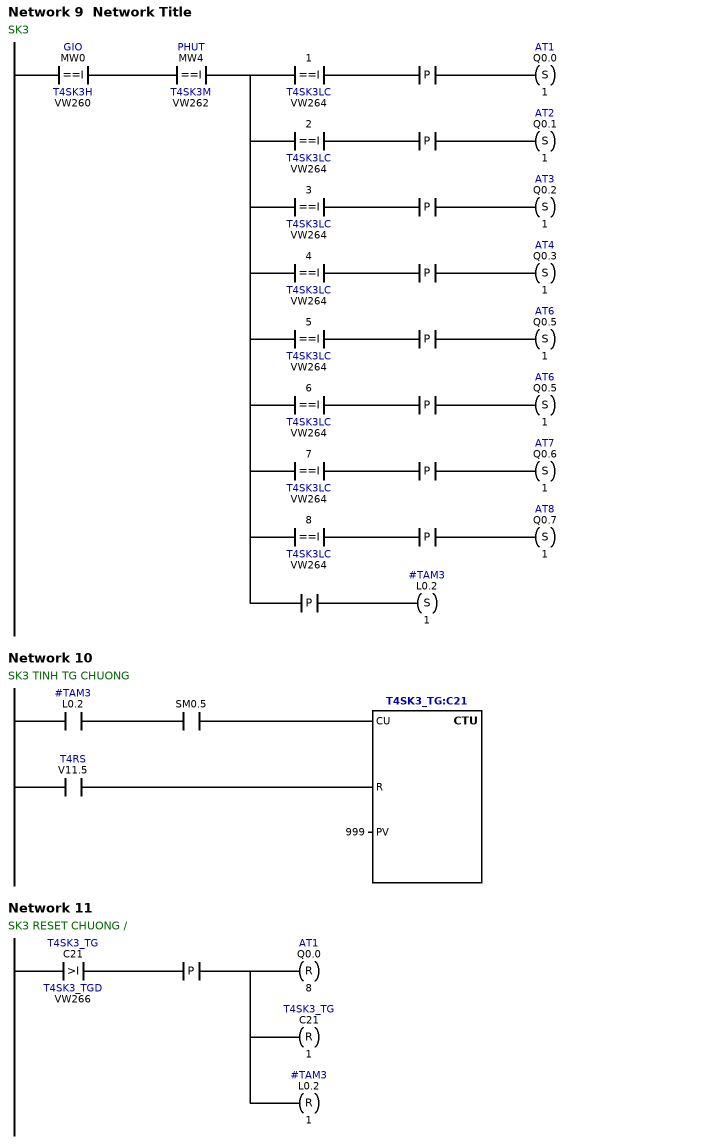
[picture p24: SBR5 networks 9-11]
Network 9 // Network Title
// SK3	
LDW=   GIO:MW0, T4SK3H:VW260
AW=    PHUT:MW4, T4SK3M:VW262
LPS
AW=    1, T4SK3LC:VW264
EU
S      AT1:Q0.0, 1
LRD
AW=    2, T4SK3LC:VW264
EU
S      AT2:Q0.1, 1
LRD
AW=    3, T4SK3LC:VW264
EU
S      AT3:Q0.2, 1
LRD
AW=    4, T4SK3LC:VW264
EU
S      AT4:Q0.3, 1
LRD
AW=    5, T4SK3LC:VW264
EU
S      AT6:Q0.5, 1
LRD
AW=    6, T4SK3LC:VW264
EU
S      AT6:Q0.5, 1
LRD
AW=    7, T4SK3LC:VW264
EU
S      AT7:Q0.6, 1
LRD
AW=    8, T4SK3LC:VW264
EU
S      AT8:Q0.7, 1
LPP
EU
S      #TAM3:L0.2, 1
Network 10
// SK3 TINH TG CHUONG
LD     #TAM3:L0.2
A      SM0.5
LD     T4RS:V11.5
CTU    T4SK3_TG:C21, 999
Network 11
// SK3 RESET CHUONG
// 
LDW>   T4SK3_TG:C21, T4SK3_TGD:VW266
EU
R      AT1:Q0.0, 8
R      T4SK3_TG:C21, 1
R      #TAM3:L0.2, 1
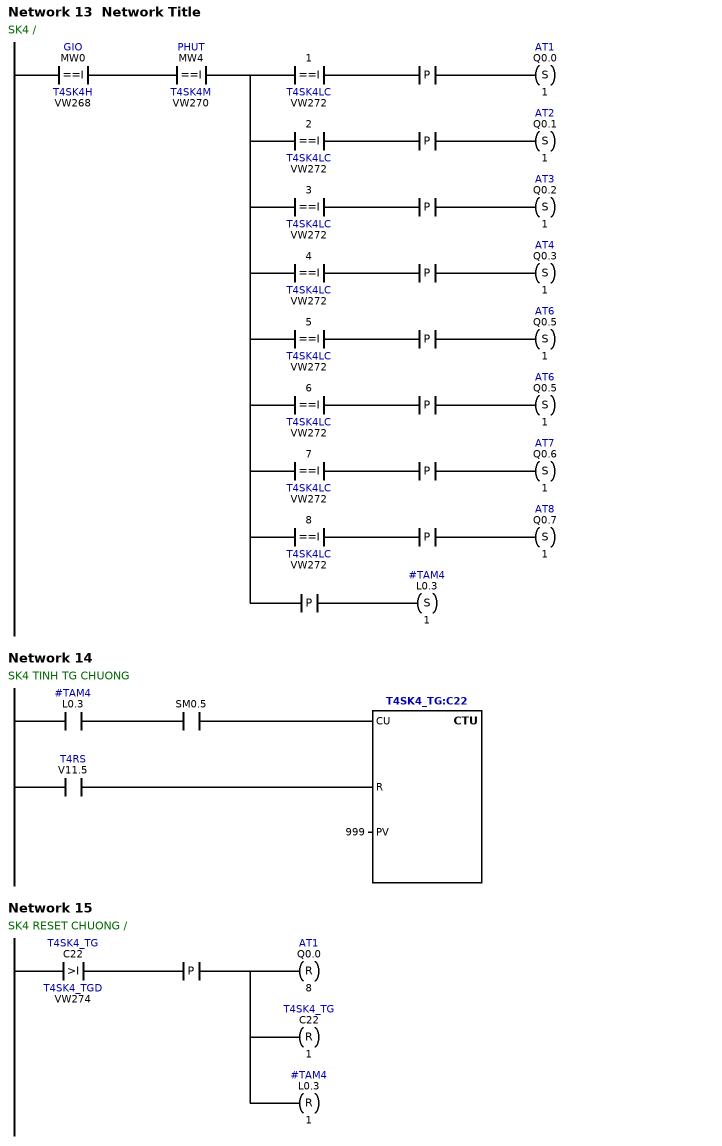
Network 13 // Network Title
// SK4
// 	
LDW=   GIO:MW0, T4SK4H:VW268
AW=    PHUT:MW4, T4SK4M:VW270
LPS
AW=    1, T4SK4LC:VW272
EU
S      AT1:Q0.0, 1
LRD
AW=    2, T4SK4LC:VW272
EU
S      AT2:Q0.1, 1
LRD
AW=    3, T4SK4LC:VW272
EU
S      AT3:Q0.2, 1
LRD
AW=    4, T4SK4LC:VW272
EU
S      AT4:Q0.3, 1
LRD
AW=    5, T4SK4LC:VW272
EU
S      AT6:Q0.5, 1
LRD
AW=    6, T4SK4LC:VW272
EU
S      AT6:Q0.5, 1
LRD
AW=    7, T4SK4LC:VW272
EU
S      AT7:Q0.6, 1
LRD
AW=    8, T4SK4LC:VW272
EU
S      AT8:Q0.7, 1
LPP
EU
S      #TAM4:L0.3, 1
Network 14
// SK4 TINH TG CHUONG
LD     #TAM4:L0.3
A      SM0.5
LD     T4RS:V11.5
CTU    T4SK4_TG:C22, 999
Network 15
// SK4 RESET CHUONG
// 
LDW>   T4SK4_TG:C22, T4SK4_TGD:VW274
EU
R      AT1:Q0.0, 8
R      T4SK4_TG:C22, 1
R      #TAM4:L0.3, 1
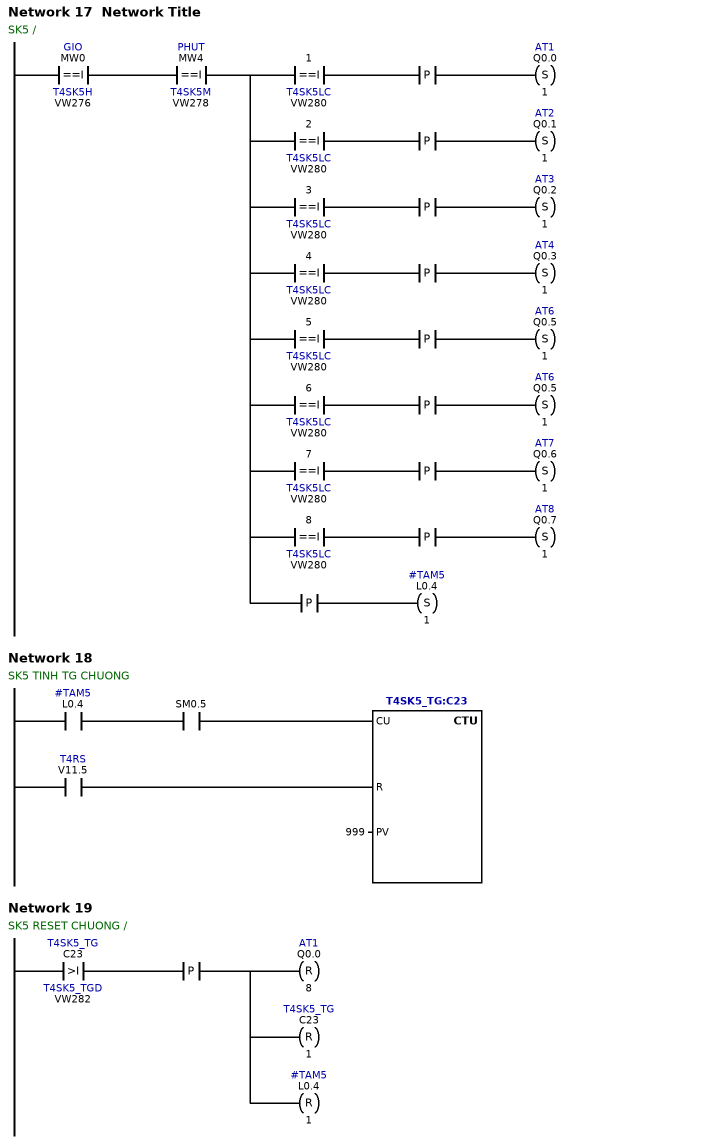
Network 17 // Network Title
// SK5
// 	
LDW=   GIO:MW0, T4SK5H:VW276
AW=    PHUT:MW4, T4SK5M:VW278
LPS
AW=    1, T4SK5LC:VW280
EU
S      AT1:Q0.0, 1
LRD
AW=    2, T4SK5LC:VW280
EU
S      AT2:Q0.1, 1
LRD
AW=    3, T4SK5LC:VW280
EU
S      AT3:Q0.2, 1
LRD
AW=    4, T4SK5LC:VW280
EU
S      AT4:Q0.3, 1
LRD
AW=    5, T4SK5LC:VW280
EU
S      AT6:Q0.5, 1
LRD
AW=    6, T4SK5LC:VW280
EU
S      AT6:Q0.5, 1
LRD
AW=    7, T4SK5LC:VW280
EU
S      AT7:Q0.6, 1
LRD
AW=    8, T4SK5LC:VW280
EU
S      AT8:Q0.7, 1
LPP
EU
S      #TAM5:L0.4, 1
Network 18
// SK5 TINH TG CHUONG
LD     #TAM5:L0.4
A      SM0.5
LD     T4RS:V11.5
CTU    T4SK5_TG:C23, 999
Network 19
// SK5 RESET CHUONG
// 
LDW>   T4SK5_TG:C23, T4SK5_TGD:VW282
EU
R      AT1:Q0.0, 8
R      T4SK5_TG:C23, 1
R      #TAM5:L0.4, 1
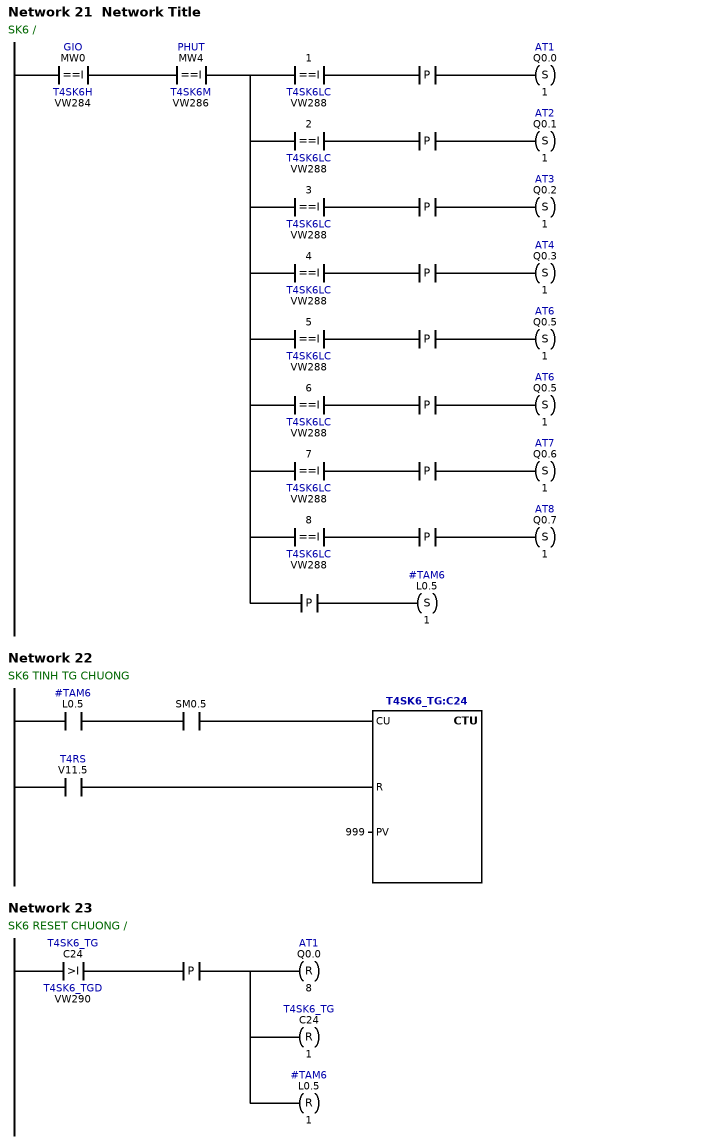
Network 21 // Network Title
// SK6
// 	
LDW=   GIO:MW0, T4SK6H:VW284
AW=    PHUT:MW4, T4SK6M:VW286
LPS
AW=    1, T4SK6LC:VW288
EU
S      AT1:Q0.0, 1
LRD
AW=    2, T4SK6LC:VW288
EU
S      AT2:Q0.1, 1
LRD
AW=    3, T4SK6LC:VW288
EU
S      AT3:Q0.2, 1
LRD
AW=    4, T4SK6LC:VW288
EU
S      AT4:Q0.3, 1
LRD
AW=    5, T4SK6LC:VW288
EU
S      AT6:Q0.5, 1
LRD
AW=    6, T4SK6LC:VW288
EU
S      AT6:Q0.5, 1
LRD
AW=    7, T4SK6LC:VW288
EU
S      AT7:Q0.6, 1
LRD
AW=    8, T4SK6LC:VW288
EU
S      AT8:Q0.7, 1
LPP
EU
S      #TAM6:L0.5, 1
Network 22
// SK6 TINH TG CHUONG
LD     #TAM6:L0.5
A      SM0.5
LD     T4RS:V11.5
CTU    T4SK6_TG:C24, 999
Network 23
// SK6 RESET CHUONG
// 
LDW>   T4SK6_TG:C24, T4SK6_TGD:VW290
EU
R      AT1:Q0.0, 8
R      T4SK6_TG:C24, 1
R      #TAM6:L0.5, 1
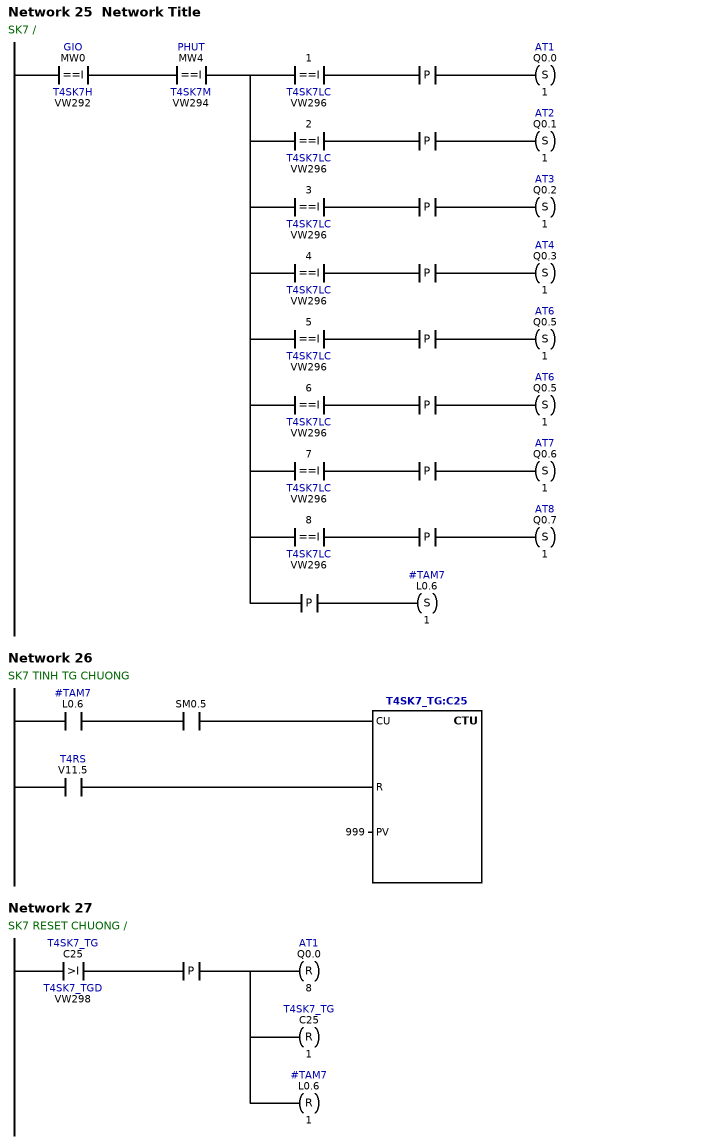
Network 25 // Network Title
// SK7
// 	
LDW=   GIO:MW0, T4SK7H:VW292
AW=    PHUT:MW4, T4SK7M:VW294
LPS
AW=    1, T4SK7LC:VW296
EU
S      AT1:Q0.0, 1
LRD
AW=    2, T4SK7LC:VW296
EU
S      AT2:Q0.1, 1
LRD
AW=    3, T4SK7LC:VW296
EU
S      AT3:Q0.2, 1
LRD
AW=    4, T4SK7LC:VW296
EU
S      AT4:Q0.3, 1
LRD
AW=    5, T4SK7LC:VW296
EU
S      AT6:Q0.5, 1
LRD
AW=    6, T4SK7LC:VW296
EU
S      AT6:Q0.5, 1
LRD
AW=    7, T4SK7LC:VW296
EU
S      AT7:Q0.6, 1
LRD
AW=    8, T4SK7LC:VW296
EU
S      AT8:Q0.7, 1
LPP
EU
S      #TAM7:L0.6, 1
Network 26
// SK7 TINH TG CHUONG
LD     #TAM7:L0.6
A      SM0.5
LD     T4RS:V11.5
CTU    T4SK7_TG:C25, 999
Network 27
// SK7 RESET CHUONG
// 
LDW>   T4SK7_TG:C25, T4SK7_TGD:VW298
EU
R      AT1:Q0.0, 8
R      T4SK7_TG:C25, 1
R      #TAM7:L0.6, 1
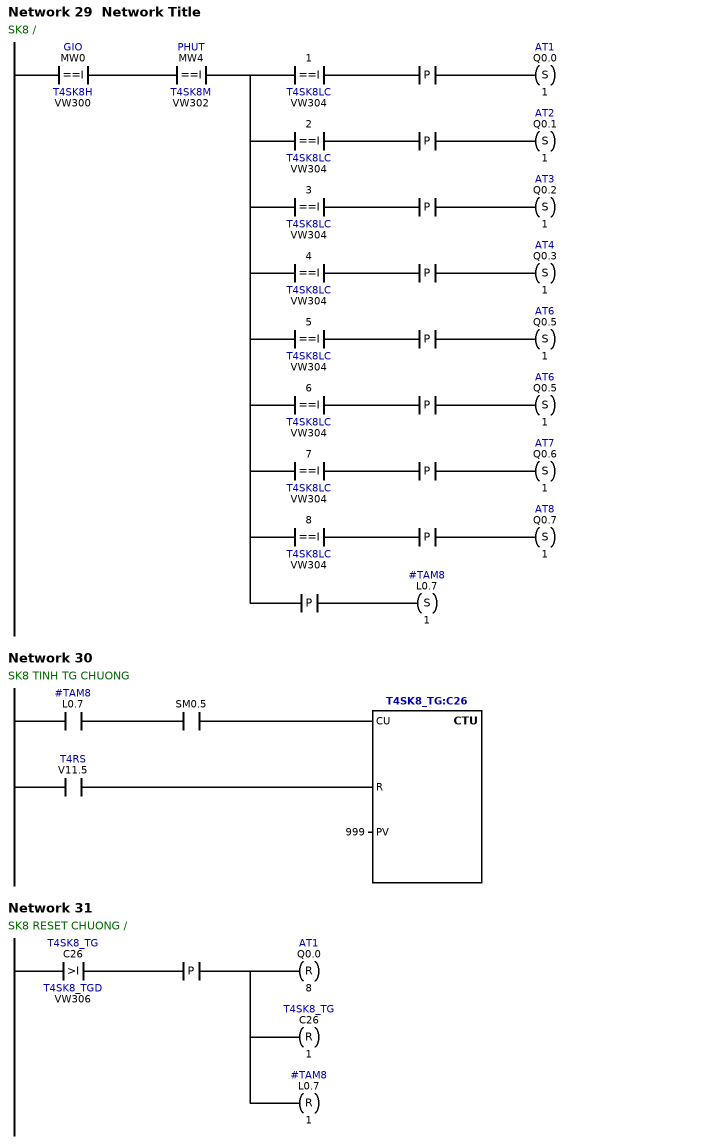
Network 29 // Network Title
// SK8
// 	
LDW=   GIO:MW0, T4SK8H:VW300
AW=    PHUT:MW4, T4SK8M:VW302
LPS
AW=    1, T4SK8LC:VW304
EU
S      AT1:Q0.0, 1
LRD
AW=    2, T4SK8LC:VW304
EU
S      AT2:Q0.1, 1
LRD
AW=    3, T4SK8LC:VW304
EU
S      AT3:Q0.2, 1
LRD
AW=    4, T4SK8LC:VW304
EU
S      AT4:Q0.3, 1
LRD
AW=    5, T4SK8LC:VW304
EU
S      AT6:Q0.5, 1
LRD
AW=    6, T4SK8LC:VW304
EU
S      AT6:Q0.5, 1
LRD
AW=    7, T4SK8LC:VW304
EU
S      AT7:Q0.6, 1
LRD
AW=    8, T4SK8LC:VW304
EU
S      AT8:Q0.7, 1
LPP
EU
S      #TAM8:L0.7, 1
Network 30
// SK8 TINH TG CHUONG
LD     #TAM8:L0.7
A      SM0.5
LD     T4RS:V11.5
CTU    T4SK8_TG:C26, 999
Network 31
// SK8 RESET CHUONG
// 
LDW>   T4SK8_TG:C26, T4SK8_TGD:VW306
EU
R      AT1:Q0.0, 8
R      T4SK8_TG:C26, 1
R      #TAM8:L0.7, 1
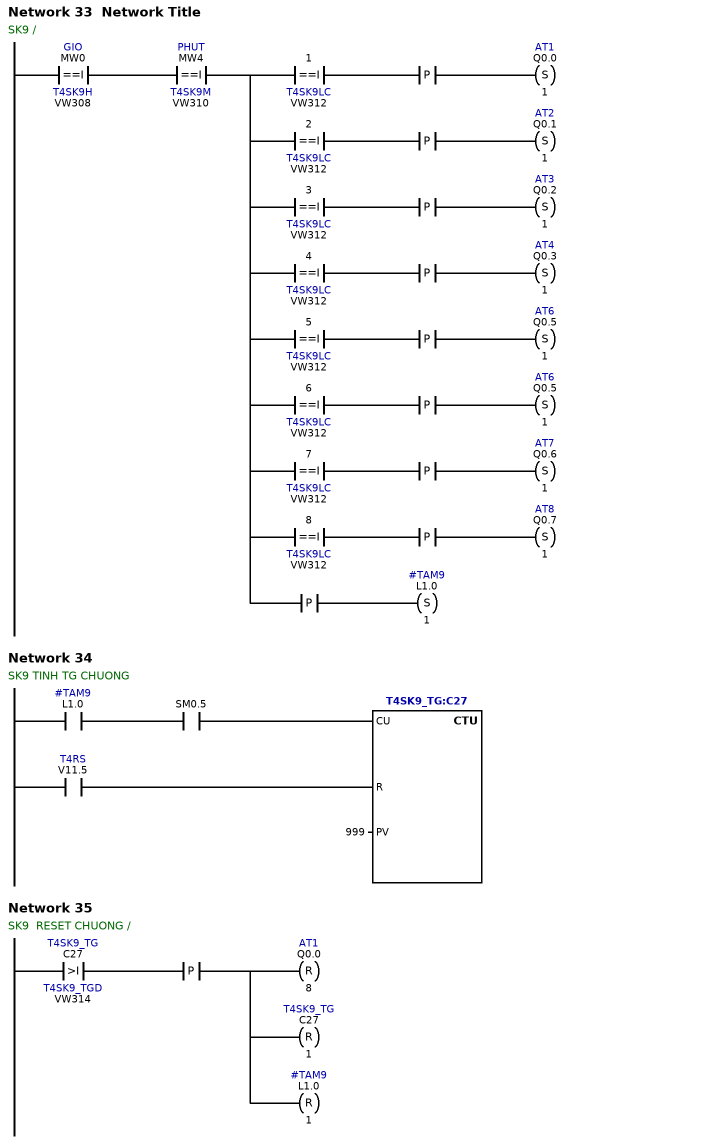
Network 33 // Network Title
// SK9
// 	
LDW=   GIO:MW0, T4SK9H:VW308
AW=    PHUT:MW4, T4SK9M:VW310
LPS
AW=    1, T4SK9LC:VW312
EU
S      AT1:Q0.0, 1
LRD
AW=    2, T4SK9LC:VW312
EU
S      AT2:Q0.1, 1
LRD
AW=    3, T4SK9LC:VW312
EU
S      AT3:Q0.2, 1
LRD
AW=    4, T4SK9LC:VW312
EU
S      AT4:Q0.3, 1
LRD
AW=    5, T4SK9LC:VW312
EU
S      AT6:Q0.5, 1
LRD
AW=    6, T4SK9LC:VW312
EU
S      AT6:Q0.5, 1
LRD
AW=    7, T4SK9LC:VW312
EU
S      AT7:Q0.6, 1
LRD
AW=    8, T4SK9LC:VW312
EU
S      AT8:Q0.7, 1
LPP
EU
S      #TAM9:L1.0, 1
Network 34
// SK9 TINH TG CHUONG
LD     #TAM9:L1.0
A      SM0.5
LD     T4RS:V11.5
CTU    T4SK9_TG:C27, 999
Network 35
// SK9  RESET CHUONG
// 
LDW>   T4SK9_TG:C27, T4SK9_TGD:VW314
EU
R      AT1:Q0.0, 8
R      T4SK9_TG:C27, 1
R      #TAM9:L1.0, 1
Network 44 // Network Title
// Network Comment
Network 54 // Network Title
// Network Comment
END_SUBROUTINE_BLOCK

SUBROUTINE_BLOCK TH5:SBR6
TITLE=SUBROUTINE COMMENTS
VAR
TAM1:BOOL;	// L0.0 
TAM2:BOOL;	// L0.1 
TAM3:BOOL;	// L0.2 
TAM4:BOOL;	// L0.3 
TAM5:BOOL;	// L0.4 
TAM6:BOOL;	// L0.5 
TAM7:BOOL;	// L0.6 
TAM8:BOOL;	// L0.7 
TAM9:BOOL;	// L1.0 
END_VAR
BEGIN
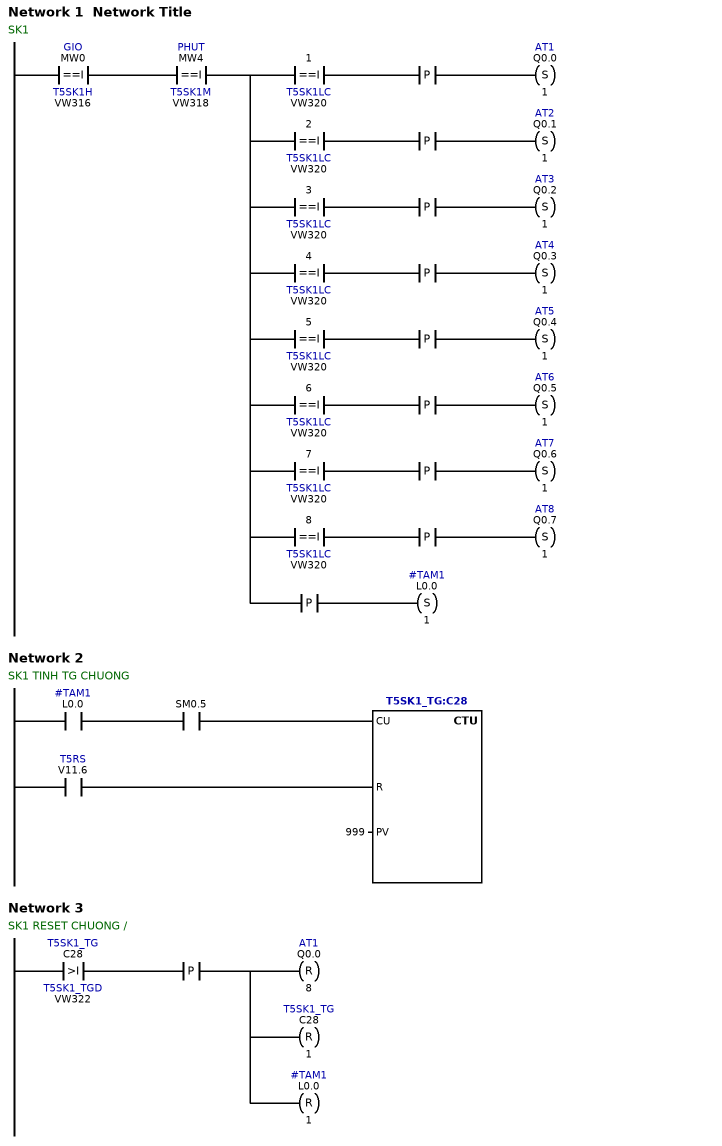
Network 1 // Network Title
// SK1	
LDW=   GIO:MW0, T5SK1H:VW316
AW=    PHUT:MW4, T5SK1M:VW318
LPS
AW=    1, T5SK1LC:VW320
EU
S      AT1:Q0.0, 1
LRD
AW=    2, T5SK1LC:VW320
EU
S      AT2:Q0.1, 1
LRD
AW=    3, T5SK1LC:VW320
EU
S      AT3:Q0.2, 1
LRD
AW=    4, T5SK1LC:VW320
EU
S      AT4:Q0.3, 1
LRD
AW=    5, T5SK1LC:VW320
EU
S      AT5:Q0.4, 1
LRD
AW=    6, T5SK1LC:VW320
EU
S      AT6:Q0.5, 1
LRD
AW=    7, T5SK1LC:VW320
EU
S      AT7:Q0.6, 1
LRD
AW=    8, T5SK1LC:VW320
EU
S      AT8:Q0.7, 1
LPP
EU
S      #TAM1:L0.0, 1
Network 2
// SK1 TINH TG CHUONG
LD     #TAM1:L0.0
A      SM0.5
LD     T5RS:V11.6
CTU    T5SK1_TG:C28, 999
Network 3
// SK1 RESET CHUONG
// 
LDW>   T5SK1_TG:C28, T5SK1_TGD:VW322
EU
R      AT1:Q0.0, 8
R      T5SK1_TG:C28, 1
R      #TAM1:L0.0, 1
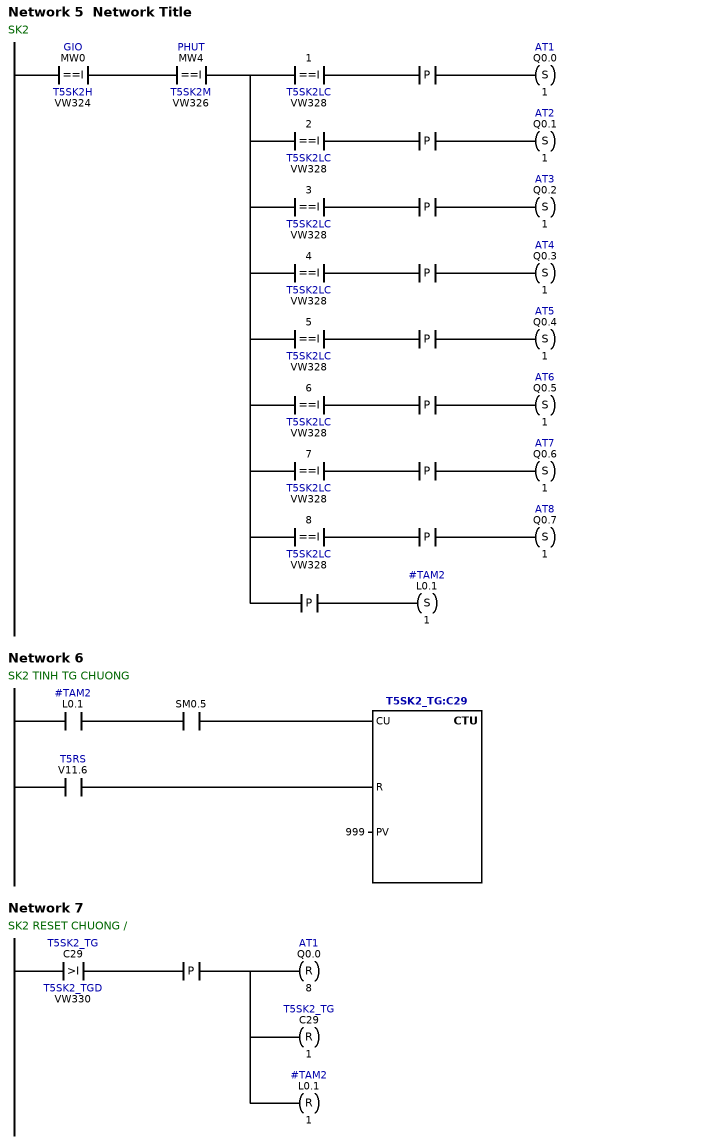
Network 5 // Network Title
// SK2
LDW=   GIO:MW0, T5SK2H:VW324
AW=    PHUT:MW4, T5SK2M:VW326
LPS
AW=    1, T5SK2LC:VW328
EU
S      AT1:Q0.0, 1
LRD
AW=    2, T5SK2LC:VW328
EU
S      AT2:Q0.1, 1
LRD
AW=    3, T5SK2LC:VW328
EU
S      AT3:Q0.2, 1
LRD
AW=    4, T5SK2LC:VW328
EU
S      AT4:Q0.3, 1
LRD
AW=    5, T5SK2LC:VW328
EU
S      AT5:Q0.4, 1
LRD
AW=    6, T5SK2LC:VW328
EU
S      AT6:Q0.5, 1
LRD
AW=    7, T5SK2LC:VW328
EU
S      AT7:Q0.6, 1
LRD
AW=    8, T5SK2LC:VW328
EU
S      AT8:Q0.7, 1
LPP
EU
S      #TAM2:L0.1, 1
Network 6
// SK2 TINH TG CHUONG
LD     #TAM2:L0.1
A      SM0.5
LD     T5RS:V11.6
CTU    T5SK2_TG:C29, 999
Network 7
// SK2 RESET CHUONG
// 
LDW>   T5SK2_TG:C29, T5SK2_TGD:VW330
EU
R      AT1:Q0.0, 8
R      T5SK2_TG:C29, 1
R      #TAM2:L0.1, 1
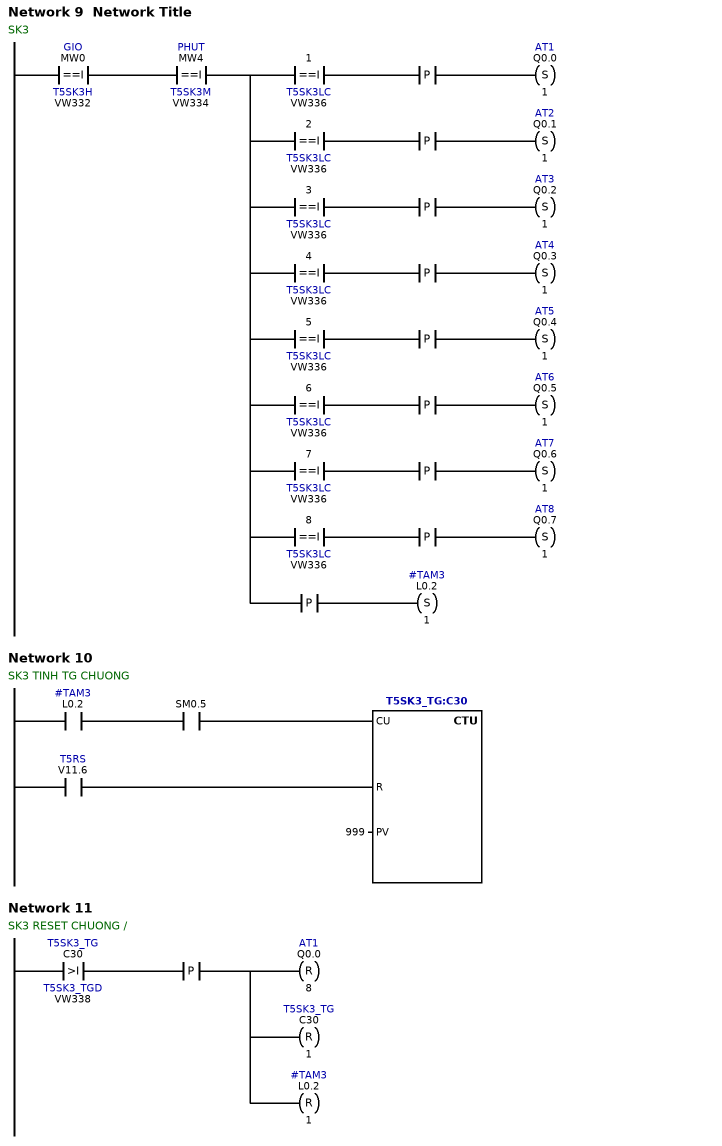
Network 9 // Network Title
// SK3	
LDW=   GIO:MW0, T5SK3H:VW332
AW=    PHUT:MW4, T5SK3M:VW334
LPS
AW=    1, T5SK3LC:VW336
EU
S      AT1:Q0.0, 1
LRD
AW=    2, T5SK3LC:VW336
EU
S      AT2:Q0.1, 1
LRD
AW=    3, T5SK3LC:VW336
EU
S      AT3:Q0.2, 1
LRD
AW=    4, T5SK3LC:VW336
EU
S      AT4:Q0.3, 1
LRD
AW=    5, T5SK3LC:VW336
EU
S      AT5:Q0.4, 1
LRD
AW=    6, T5SK3LC:VW336
EU
S      AT6:Q0.5, 1
LRD
AW=    7, T5SK3LC:VW336
EU
S      AT7:Q0.6, 1
LRD
AW=    8, T5SK3LC:VW336
EU
S      AT8:Q0.7, 1
LPP
EU
S      #TAM3:L0.2, 1
Network 10
// SK3 TINH TG CHUONG
LD     #TAM3:L0.2
A      SM0.5
LD     T5RS:V11.6
CTU    T5SK3_TG:C30, 999
Network 11
// SK3 RESET CHUONG
// 
LDW>   T5SK3_TG:C30, T5SK3_TGD:VW338
EU
R      AT1:Q0.0, 8
R      T5SK3_TG:C30, 1
R      #TAM3:L0.2, 1
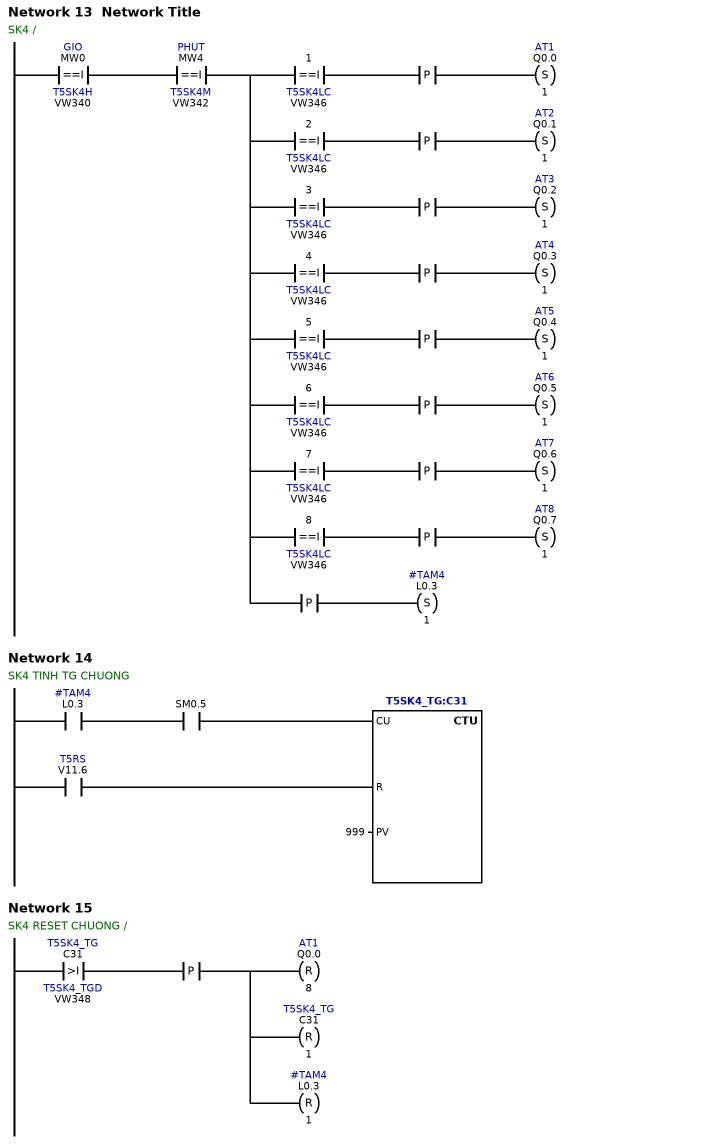
Network 13 // Network Title
// SK4
// 	
LDW=   GIO:MW0, T5SK4H:VW340
AW=    PHUT:MW4, T5SK4M:VW342
LPS
AW=    1, T5SK4LC:VW346
EU
S      AT1:Q0.0, 1
LRD
AW=    2, T5SK4LC:VW346
EU
S      AT2:Q0.1, 1
LRD
AW=    3, T5SK4LC:VW346
EU
S      AT3:Q0.2, 1
LRD
AW=    4, T5SK4LC:VW346
EU
S      AT4:Q0.3, 1
LRD
AW=    5, T5SK4LC:VW346
EU
S      AT5:Q0.4, 1
LRD
AW=    6, T5SK4LC:VW346
EU
S      AT6:Q0.5, 1
LRD
AW=    7, T5SK4LC:VW346
EU
S      AT7:Q0.6, 1
LRD
AW=    8, T5SK4LC:VW346
EU
S      AT8:Q0.7, 1
LPP
EU
S      #TAM4:L0.3, 1
Network 14
// SK4 TINH TG CHUONG
LD     #TAM4:L0.3
A      SM0.5
LD     T5RS:V11.6
CTU    T5SK4_TG:C31, 999
Network 15
// SK4 RESET CHUONG
// 
LDW>   T5SK4_TG:C31, T5SK4_TGD:VW348
EU
R      AT1:Q0.0, 8
R      T5SK4_TG:C31, 1
R      #TAM4:L0.3, 1
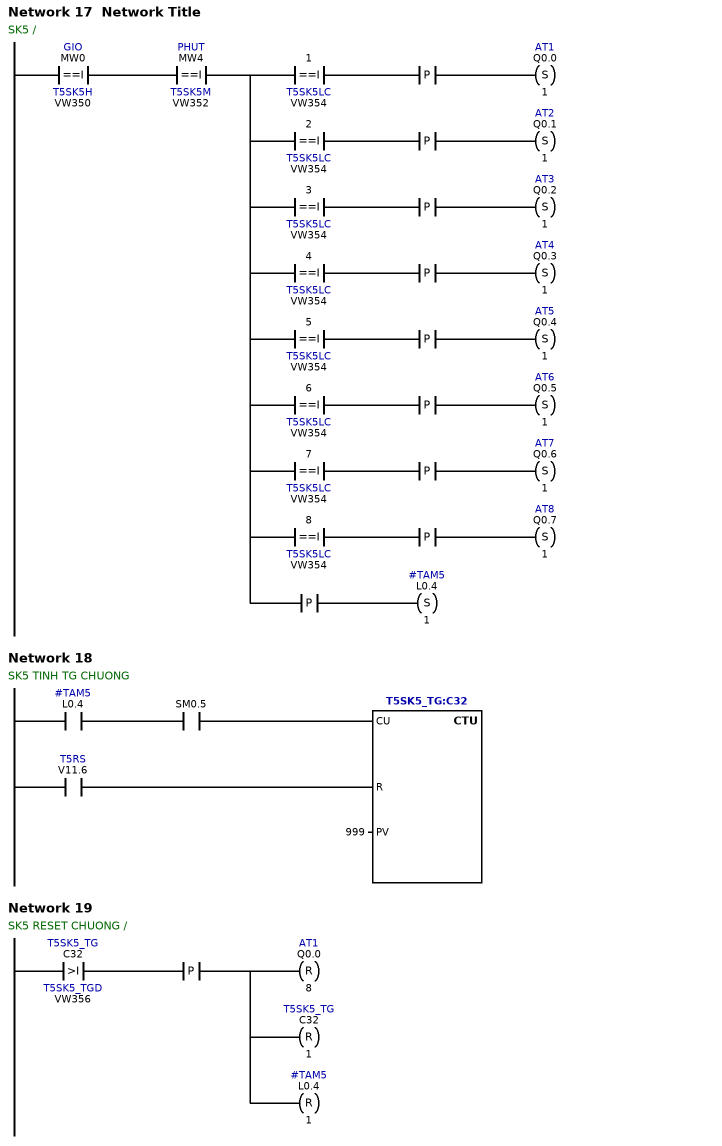
Network 17 // Network Title
// SK5
// 	
LDW=   GIO:MW0, T5SK5H:VW350
AW=    PHUT:MW4, T5SK5M:VW352
LPS
AW=    1, T5SK5LC:VW354
EU
S      AT1:Q0.0, 1
LRD
AW=    2, T5SK5LC:VW354
EU
S      AT2:Q0.1, 1
LRD
AW=    3, T5SK5LC:VW354
EU
S      AT3:Q0.2, 1
LRD
AW=    4, T5SK5LC:VW354
EU
S      AT4:Q0.3, 1
LRD
AW=    5, T5SK5LC:VW354
EU
S      AT5:Q0.4, 1
LRD
AW=    6, T5SK5LC:VW354
EU
S      AT6:Q0.5, 1
LRD
AW=    7, T5SK5LC:VW354
EU
S      AT7:Q0.6, 1
LRD
AW=    8, T5SK5LC:VW354
EU
S      AT8:Q0.7, 1
LPP
EU
S      #TAM5:L0.4, 1
Network 18
// SK5 TINH TG CHUONG
LD     #TAM5:L0.4
A      SM0.5
LD     T5RS:V11.6
CTU    T5SK5_TG:C32, 999
Network 19
// SK5 RESET CHUONG
// 
LDW>   T5SK5_TG:C32, T5SK5_TGD:VW356
EU
R      AT1:Q0.0, 8
R      T5SK5_TG:C32, 1
R      #TAM5:L0.4, 1
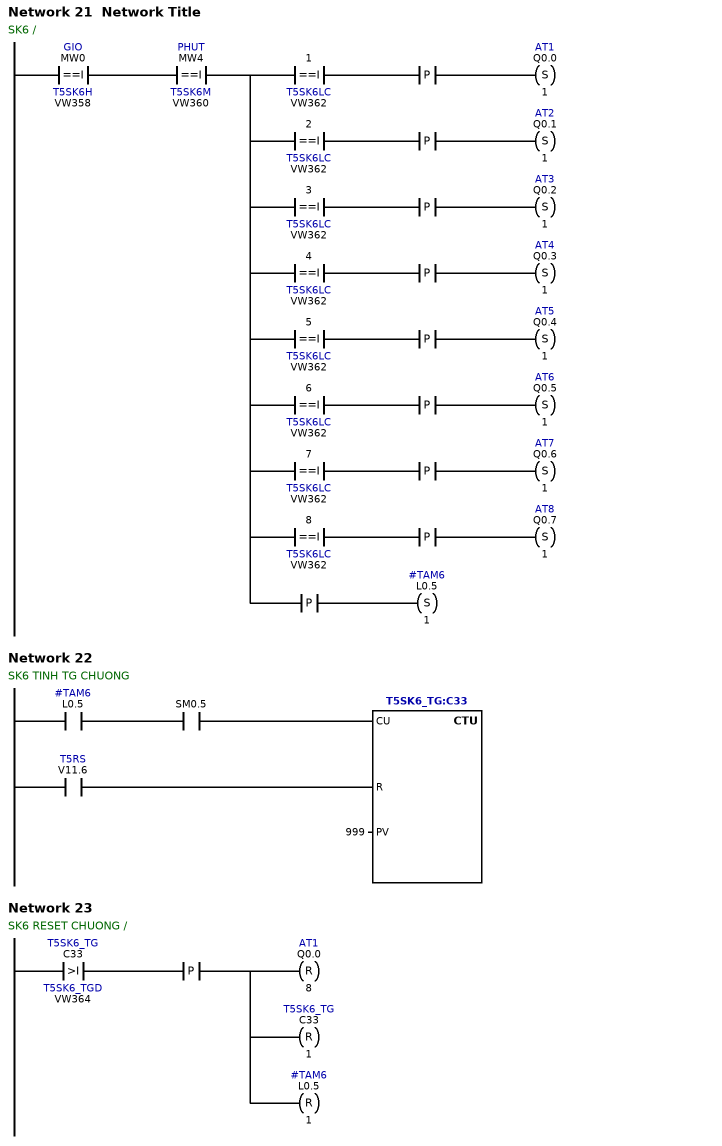
Network 21 // Network Title
// SK6
// 	
LDW=   GIO:MW0, T5SK6H:VW358
AW=    PHUT:MW4, T5SK6M:VW360
LPS
AW=    1, T5SK6LC:VW362
EU
S      AT1:Q0.0, 1
LRD
AW=    2, T5SK6LC:VW362
EU
S      AT2:Q0.1, 1
LRD
AW=    3, T5SK6LC:VW362
EU
S      AT3:Q0.2, 1
LRD
AW=    4, T5SK6LC:VW362
EU
S      AT4:Q0.3, 1
LRD
AW=    5, T5SK6LC:VW362
EU
S      AT5:Q0.4, 1
LRD
AW=    6, T5SK6LC:VW362
EU
S      AT6:Q0.5, 1
LRD
AW=    7, T5SK6LC:VW362
EU
S      AT7:Q0.6, 1
LRD
AW=    8, T5SK6LC:VW362
EU
S      AT8:Q0.7, 1
LPP
EU
S      #TAM6:L0.5, 1
Network 22
// SK6 TINH TG CHUONG
LD     #TAM6:L0.5
A      SM0.5
LD     T5RS:V11.6
CTU    T5SK6_TG:C33, 999
Network 23
// SK6 RESET CHUONG
// 
LDW>   T5SK6_TG:C33, T5SK6_TGD:VW364
EU
R      AT1:Q0.0, 8
R      T5SK6_TG:C33, 1
R      #TAM6:L0.5, 1
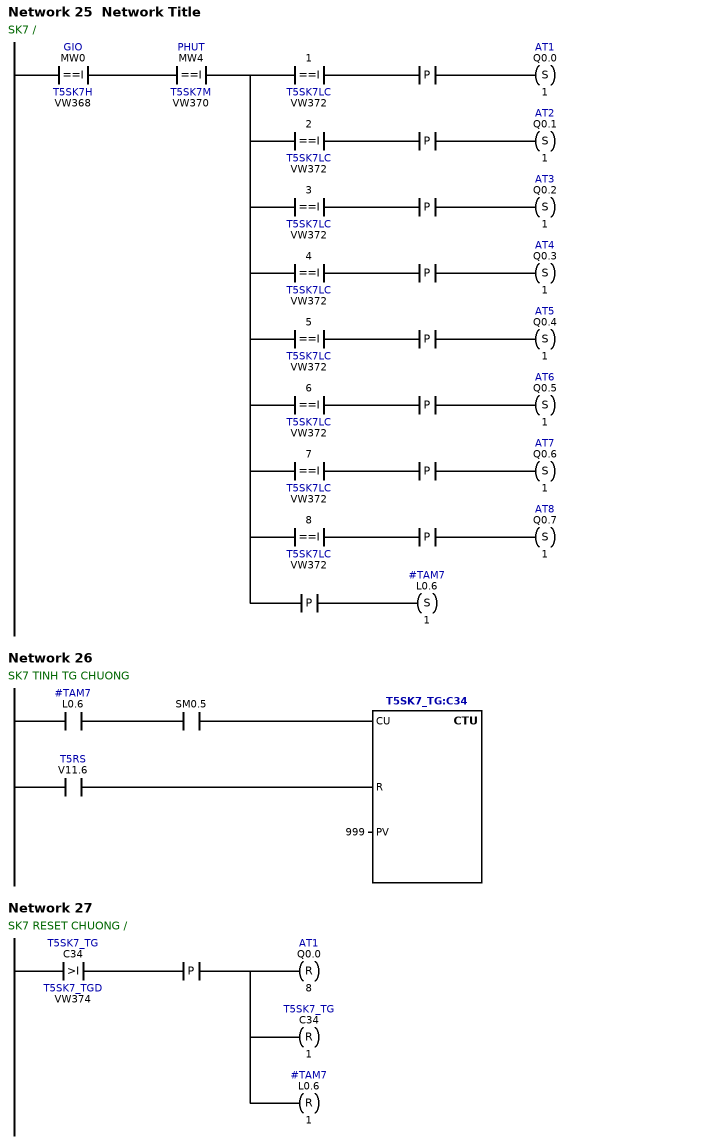
Network 25 // Network Title
// SK7
// 	
LDW=   GIO:MW0, T5SK7H:VW368
AW=    PHUT:MW4, T5SK7M:VW370
LPS
AW=    1, T5SK7LC:VW372
EU
S      AT1:Q0.0, 1
LRD
AW=    2, T5SK7LC:VW372
EU
S      AT2:Q0.1, 1
LRD
AW=    3, T5SK7LC:VW372
EU
S      AT3:Q0.2, 1
LRD
AW=    4, T5SK7LC:VW372
EU
S      AT4:Q0.3, 1
LRD
AW=    5, T5SK7LC:VW372
EU
S      AT5:Q0.4, 1
LRD
AW=    6, T5SK7LC:VW372
EU
S      AT6:Q0.5, 1
LRD
AW=    7, T5SK7LC:VW372
EU
S      AT7:Q0.6, 1
LRD
AW=    8, T5SK7LC:VW372
EU
S      AT8:Q0.7, 1
LPP
EU
S      #TAM7:L0.6, 1
Network 26
// SK7 TINH TG CHUONG
LD     #TAM7:L0.6
A      SM0.5
LD     T5RS:V11.6
CTU    T5SK7_TG:C34, 999
Network 27
// SK7 RESET CHUONG
// 
LDW>   T5SK7_TG:C34, T5SK7_TGD:VW374
EU
R      AT1:Q0.0, 8
R      T5SK7_TG:C34, 1
R      #TAM7:L0.6, 1
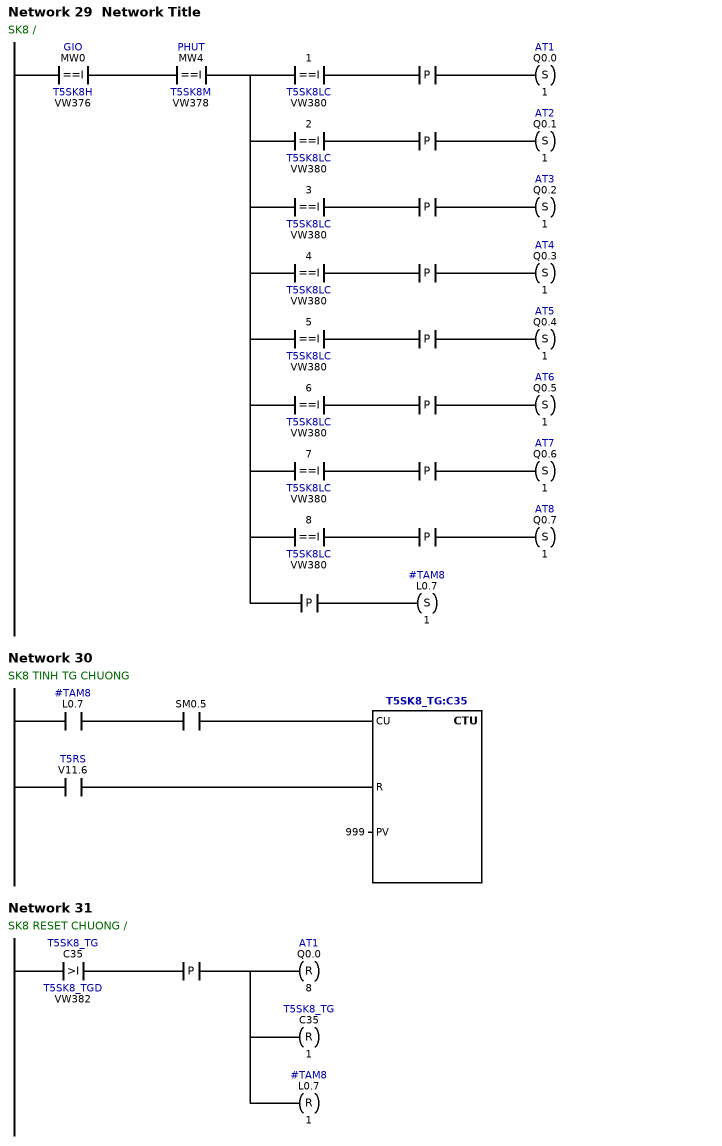
Network 29 // Network Title
// SK8
// 	
LDW=   GIO:MW0, T5SK8H:VW376
AW=    PHUT:MW4, T5SK8M:VW378
LPS
AW=    1, T5SK8LC:VW380
EU
S      AT1:Q0.0, 1
LRD
AW=    2, T5SK8LC:VW380
EU
S      AT2:Q0.1, 1
LRD
AW=    3, T5SK8LC:VW380
EU
S      AT3:Q0.2, 1
LRD
AW=    4, T5SK8LC:VW380
EU
S      AT4:Q0.3, 1
LRD
AW=    5, T5SK8LC:VW380
EU
S      AT5:Q0.4, 1
LRD
AW=    6, T5SK8LC:VW380
EU
S      AT6:Q0.5, 1
LRD
AW=    7, T5SK8LC:VW380
EU
S      AT7:Q0.6, 1
LRD
AW=    8, T5SK8LC:VW380
EU
S      AT8:Q0.7, 1
LPP
EU
S      #TAM8:L0.7, 1
Network 30
// SK8 TINH TG CHUONG
LD     #TAM8:L0.7
A      SM0.5
LD     T5RS:V11.6
CTU    T5SK8_TG:C35, 999
Network 31
// SK8 RESET CHUONG
// 
LDW>   T5SK8_TG:C35, T5SK8_TGD:VW382
EU
R      AT1:Q0.0, 8
R      T5SK8_TG:C35, 1
R      #TAM8:L0.7, 1
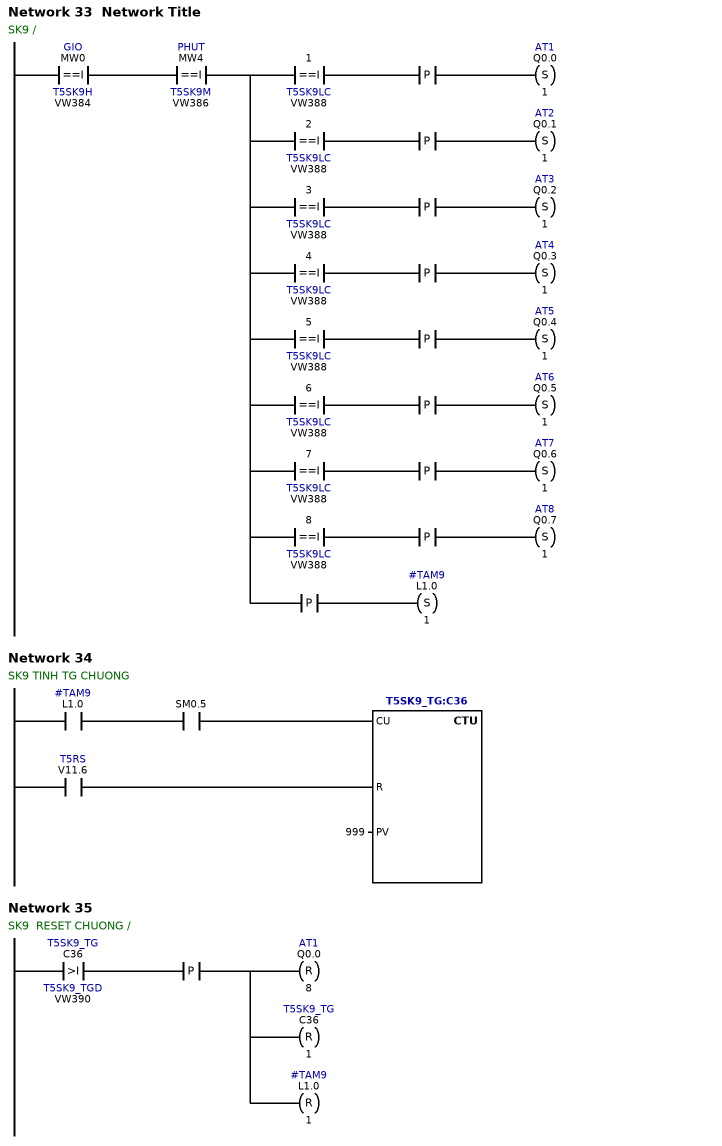
Network 33 // Network Title
// SK9
// 	
LDW=   GIO:MW0, T5SK9H:VW384
AW=    PHUT:MW4, T5SK9M:VW386
LPS
AW=    1, T5SK9LC:VW388
EU
S      AT1:Q0.0, 1
LRD
AW=    2, T5SK9LC:VW388
EU
S      AT2:Q0.1, 1
LRD
AW=    3, T5SK9LC:VW388
EU
S      AT3:Q0.2, 1
LRD
AW=    4, T5SK9LC:VW388
EU
S      AT4:Q0.3, 1
LRD
AW=    5, T5SK9LC:VW388
EU
S      AT5:Q0.4, 1
LRD
AW=    6, T5SK9LC:VW388
EU
S      AT6:Q0.5, 1
LRD
AW=    7, T5SK9LC:VW388
EU
S      AT7:Q0.6, 1
LRD
AW=    8, T5SK9LC:VW388
EU
S      AT8:Q0.7, 1
LPP
EU
S      #TAM9:L1.0, 1
Network 34
// SK9 TINH TG CHUONG
LD     #TAM9:L1.0
A      SM0.5
LD     T5RS:V11.6
CTU    T5SK9_TG:C36, 999
Network 35
// SK9  RESET CHUONG
// 
LDW>   T5SK9_TG:C36, T5SK9_TGD:VW390
EU
R      AT1:Q0.0, 8
R      T5SK9_TG:C36, 1
R      #TAM9:L1.0, 1
Network 44 // Network Title
// Network Comment
Network 54 // Network Title
// Network Comment
Network 64 // Network Title
// Network Comment
END_SUBROUTINE_BLOCK

SUBROUTINE_BLOCK TH6:SBR7
TITLE=SUBROUTINE COMMENTS
VAR
TAM1:BOOL;	// L0.0 
TAM2:BOOL;	// L0.1 
TAM3:BOOL;	// L0.2 
TAM4:BOOL;	// L0.3 
TAM5:BOOL;	// L0.4 
TAM6:BOOL;	// L0.5 
TAM7:BOOL;	// L0.6 
TAM8:BOOL;	// L0.7 
TAM9:BOOL;	// L1.0 
END_VAR
BEGIN
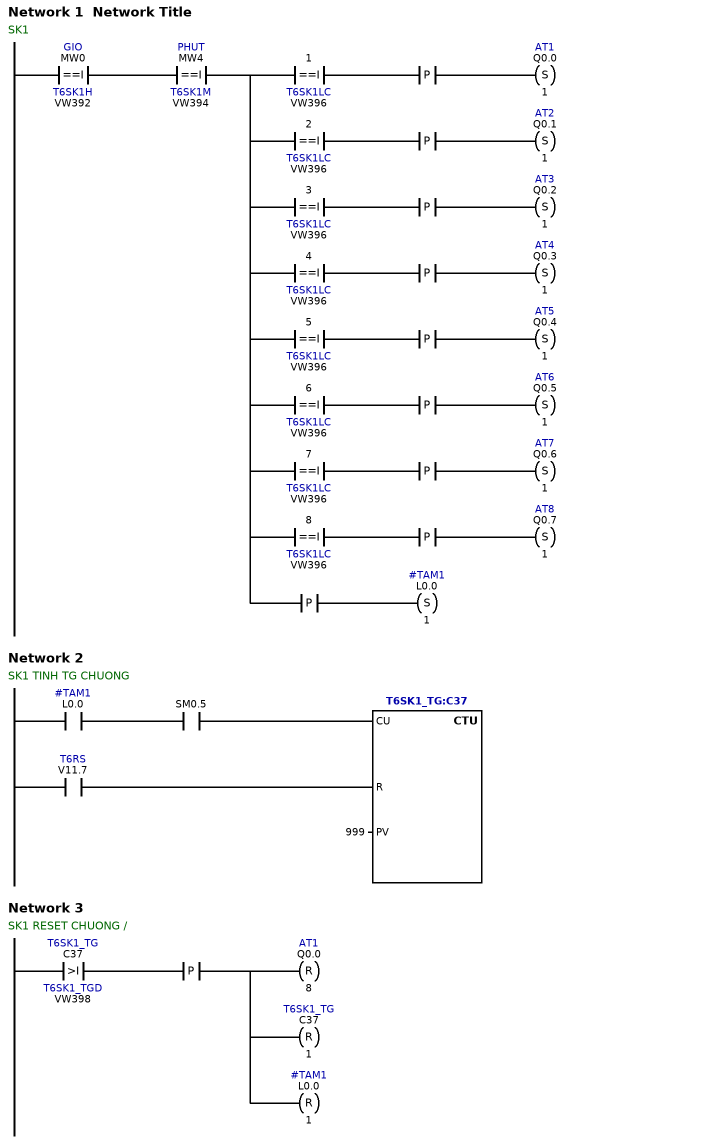
Network 1 // Network Title
// SK1	
LDW=   GIO:MW0, T6SK1H:VW392
AW=    PHUT:MW4, T6SK1M:VW394
LPS
AW=    1, T6SK1LC:VW396
EU
S      AT1:Q0.0, 1
LRD
AW=    2, T6SK1LC:VW396
EU
S      AT2:Q0.1, 1
LRD
AW=    3, T6SK1LC:VW396
EU
S      AT3:Q0.2, 1
LRD
AW=    4, T6SK1LC:VW396
EU
S      AT4:Q0.3, 1
LRD
AW=    5, T6SK1LC:VW396
EU
S      AT5:Q0.4, 1
LRD
AW=    6, T6SK1LC:VW396
EU
S      AT6:Q0.5, 1
LRD
AW=    7, T6SK1LC:VW396
EU
S      AT7:Q0.6, 1
LRD
AW=    8, T6SK1LC:VW396
EU
S      AT8:Q0.7, 1
LPP
EU
S      #TAM1:L0.0, 1
Network 2
// SK1 TINH TG CHUONG
LD     #TAM1:L0.0
A      SM0.5
LD     T6RS:V11.7
CTU    T6SK1_TG:C37, 999
Network 3
// SK1 RESET CHUONG
// 
LDW>   T6SK1_TG:C37, T6SK1_TGD:VW398
EU
R      AT1:Q0.0, 8
R      T6SK1_TG:C37, 1
R      #TAM1:L0.0, 1
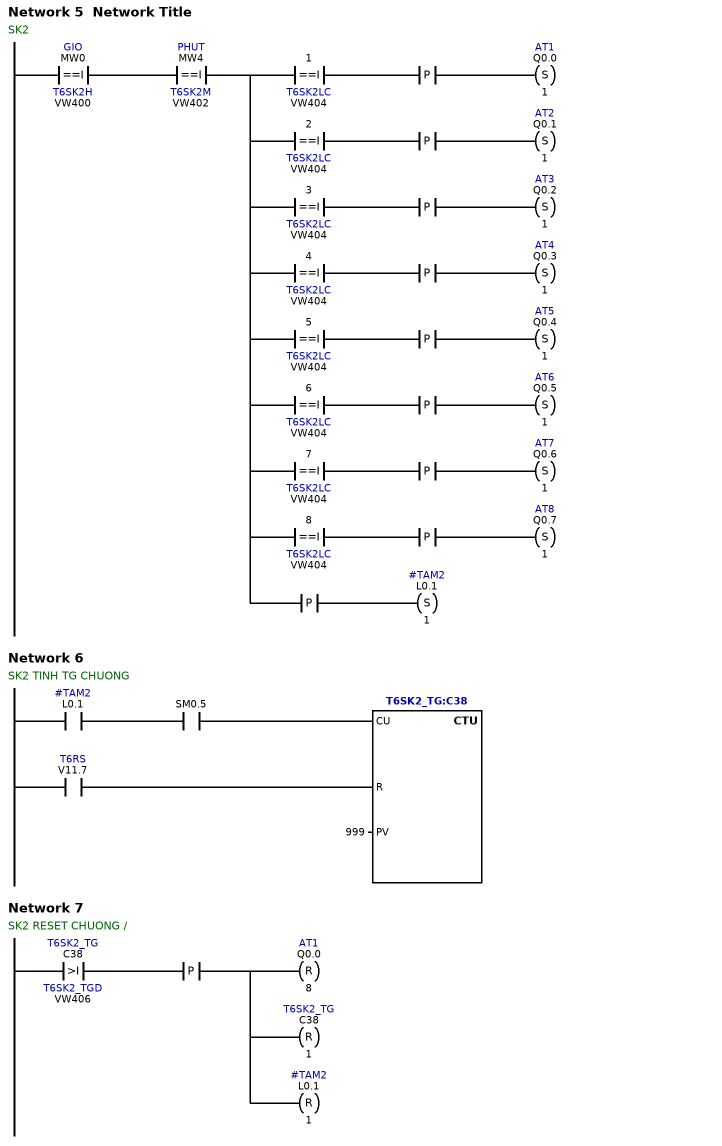
Network 5 // Network Title
// SK2
LDW=   GIO:MW0, T6SK2H:VW400
AW=    PHUT:MW4, T6SK2M:VW402
LPS
AW=    1, T6SK2LC:VW404
EU
S      AT1:Q0.0, 1
LRD
AW=    2, T6SK2LC:VW404
EU
S      AT2:Q0.1, 1
LRD
AW=    3, T6SK2LC:VW404
EU
S      AT3:Q0.2, 1
LRD
AW=    4, T6SK2LC:VW404
EU
S      AT4:Q0.3, 1
LRD
AW=    5, T6SK2LC:VW404
EU
S      AT5:Q0.4, 1
LRD
AW=    6, T6SK2LC:VW404
EU
S      AT6:Q0.5, 1
LRD
AW=    7, T6SK2LC:VW404
EU
S      AT7:Q0.6, 1
LRD
AW=    8, T6SK2LC:VW404
EU
S      AT8:Q0.7, 1
LPP
EU
S      #TAM2:L0.1, 1
Network 6
// SK2 TINH TG CHUONG
LD     #TAM2:L0.1
A      SM0.5
LD     T6RS:V11.7
CTU    T6SK2_TG:C38, 999
Network 7
// SK2 RESET CHUONG
// 
LDW>   T6SK2_TG:C38, T6SK2_TGD:VW406
EU
R      AT1:Q0.0, 8
R      T6SK2_TG:C38, 1
R      #TAM2:L0.1, 1
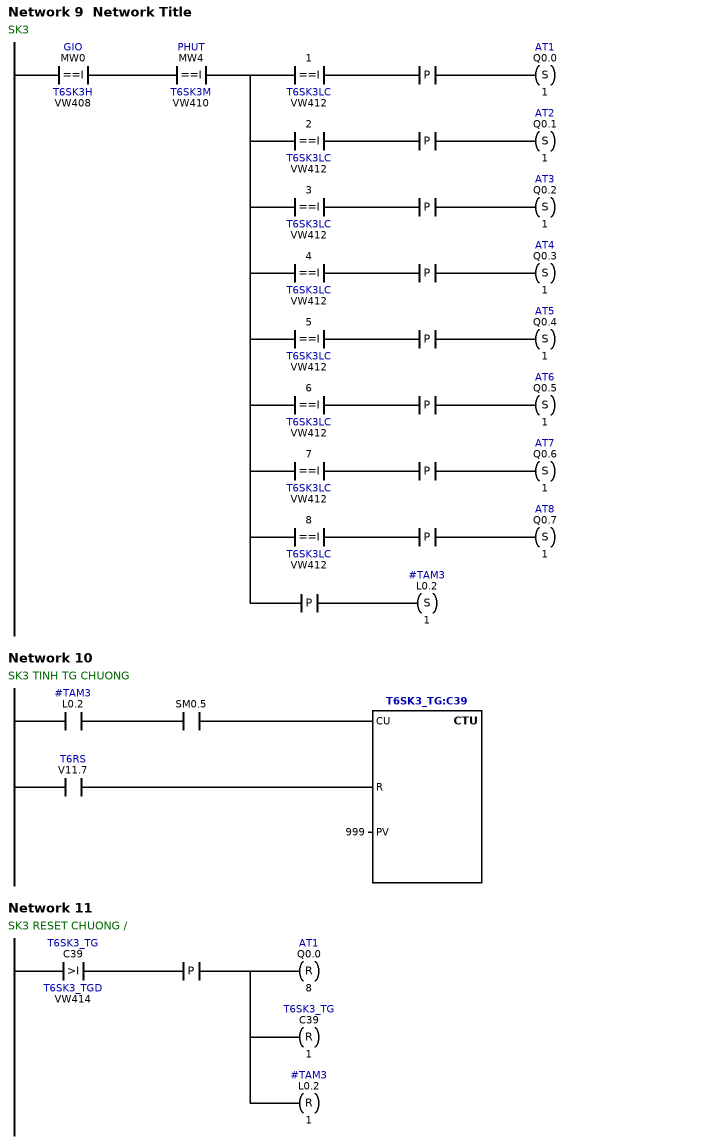
Network 9 // Network Title
// SK3	
LDW=   GIO:MW0, T6SK3H:VW408
AW=    PHUT:MW4, T6SK3M:VW410
LPS
AW=    1, T6SK3LC:VW412
EU
S      AT1:Q0.0, 1
LRD
AW=    2, T6SK3LC:VW412
EU
S      AT2:Q0.1, 1
LRD
AW=    3, T6SK3LC:VW412
EU
S      AT3:Q0.2, 1
LRD
AW=    4, T6SK3LC:VW412
EU
S      AT4:Q0.3, 1
LRD
AW=    5, T6SK3LC:VW412
EU
S      AT5:Q0.4, 1
LRD
AW=    6, T6SK3LC:VW412
EU
S      AT6:Q0.5, 1
LRD
AW=    7, T6SK3LC:VW412
EU
S      AT7:Q0.6, 1
LRD
AW=    8, T6SK3LC:VW412
EU
S      AT8:Q0.7, 1
LPP
EU
S      #TAM3:L0.2, 1
Network 10
// SK3 TINH TG CHUONG
LD     #TAM3:L0.2
A      SM0.5
LD     T6RS:V11.7
CTU    T6SK3_TG:C39, 999
Network 11
// SK3 RESET CHUONG
// 
LDW>   T6SK3_TG:C39, T6SK3_TGD:VW414
EU
R      AT1:Q0.0, 8
R      T6SK3_TG:C39, 1
R      #TAM3:L0.2, 1
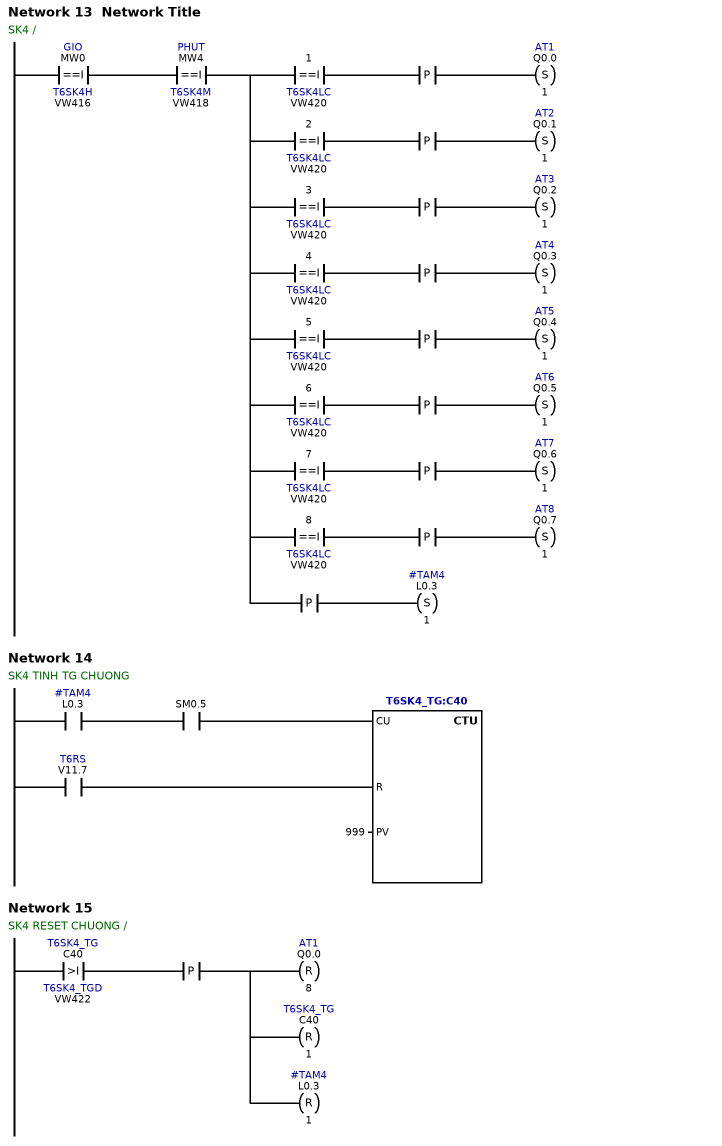
Network 13 // Network Title
// SK4
// 	
LDW=   GIO:MW0, T6SK4H:VW416
AW=    PHUT:MW4, T6SK4M:VW418
LPS
AW=    1, T6SK4LC:VW420
EU
S      AT1:Q0.0, 1
LRD
AW=    2, T6SK4LC:VW420
EU
S      AT2:Q0.1, 1
LRD
AW=    3, T6SK4LC:VW420
EU
S      AT3:Q0.2, 1
LRD
AW=    4, T6SK4LC:VW420
EU
S      AT4:Q0.3, 1
LRD
AW=    5, T6SK4LC:VW420
EU
S      AT5:Q0.4, 1
LRD
AW=    6, T6SK4LC:VW420
EU
S      AT6:Q0.5, 1
LRD
AW=    7, T6SK4LC:VW420
EU
S      AT7:Q0.6, 1
LRD
AW=    8, T6SK4LC:VW420
EU
S      AT8:Q0.7, 1
LPP
EU
S      #TAM4:L0.3, 1
Network 14
// SK4 TINH TG CHUONG
LD     #TAM4:L0.3
A      SM0.5
LD     T6RS:V11.7
CTU    T6SK4_TG:C40, 999
Network 15
// SK4 RESET CHUONG
// 
LDW>   T6SK4_TG:C40, T6SK4_TGD:VW422
EU
R      AT1:Q0.0, 8
R      T6SK4_TG:C40, 1
R      #TAM4:L0.3, 1
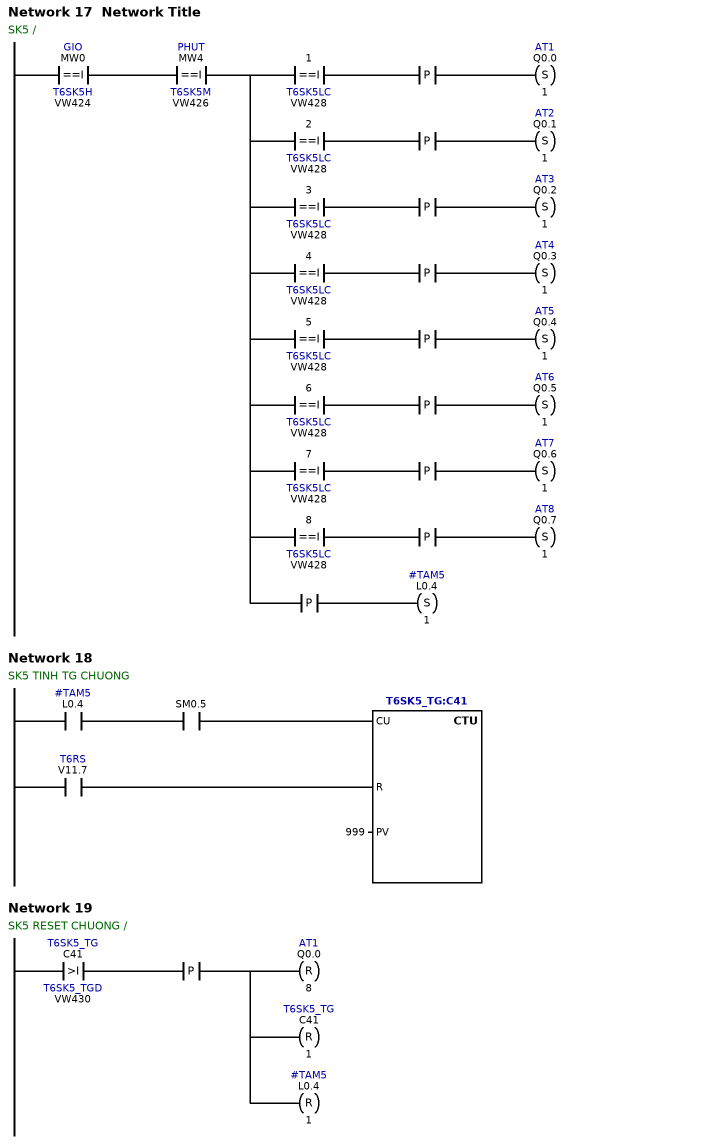
Network 17 // Network Title
// SK5
// 	
LDW=   GIO:MW0, T6SK5H:VW424
AW=    PHUT:MW4, T6SK5M:VW426
LPS
AW=    1, T6SK5LC:VW428
EU
S      AT1:Q0.0, 1
LRD
AW=    2, T6SK5LC:VW428
EU
S      AT2:Q0.1, 1
LRD
AW=    3, T6SK5LC:VW428
EU
S      AT3:Q0.2, 1
LRD
AW=    4, T6SK5LC:VW428
EU
S      AT4:Q0.3, 1
LRD
AW=    5, T6SK5LC:VW428
EU
S      AT5:Q0.4, 1
LRD
AW=    6, T6SK5LC:VW428
EU
S      AT6:Q0.5, 1
LRD
AW=    7, T6SK5LC:VW428
EU
S      AT7:Q0.6, 1
LRD
AW=    8, T6SK5LC:VW428
EU
S      AT8:Q0.7, 1
LPP
EU
S      #TAM5:L0.4, 1
Network 18
// SK5 TINH TG CHUONG
LD     #TAM5:L0.4
A      SM0.5
LD     T6RS:V11.7
CTU    T6SK5_TG:C41, 999
Network 19
// SK5 RESET CHUONG
// 
LDW>   T6SK5_TG:C41, T6SK5_TGD:VW430
EU
R      AT1:Q0.0, 8
R      T6SK5_TG:C41, 1
R      #TAM5:L0.4, 1
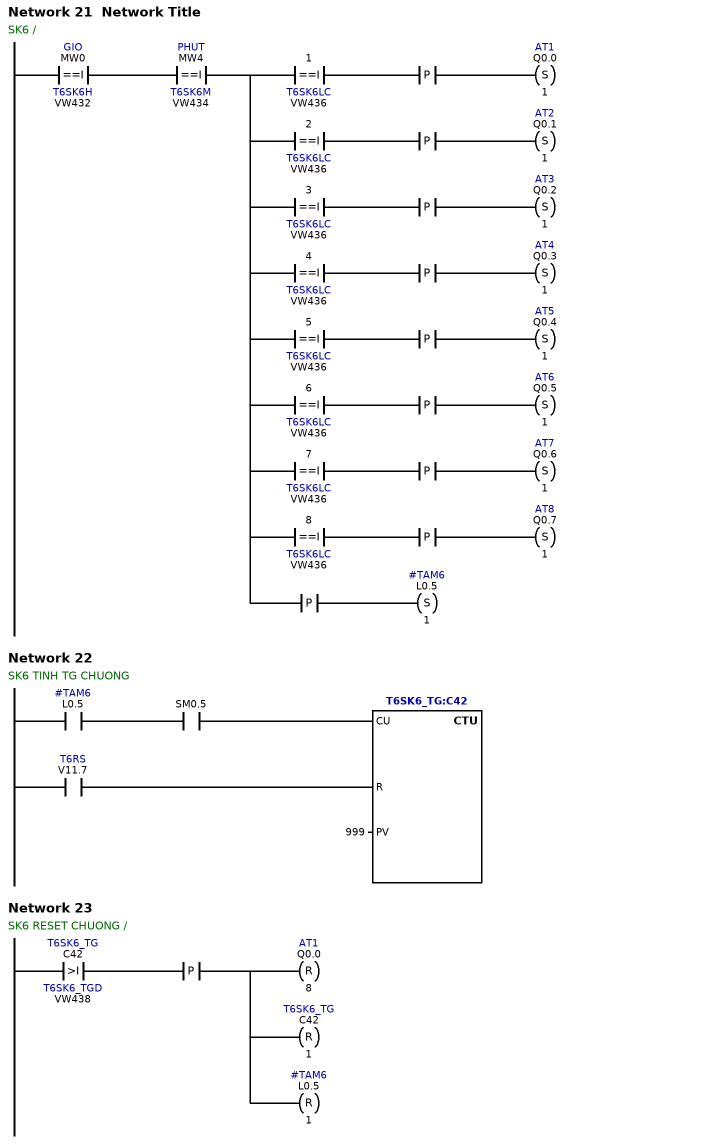
Network 21 // Network Title
// SK6
// 	
LDW=   GIO:MW0, T6SK6H:VW432
AW=    PHUT:MW4, T6SK6M:VW434
LPS
AW=    1, T6SK6LC:VW436
EU
S      AT1:Q0.0, 1
LRD
AW=    2, T6SK6LC:VW436
EU
S      AT2:Q0.1, 1
LRD
AW=    3, T6SK6LC:VW436
EU
S      AT3:Q0.2, 1
LRD
AW=    4, T6SK6LC:VW436
EU
S      AT4:Q0.3, 1
LRD
AW=    5, T6SK6LC:VW436
EU
S      AT5:Q0.4, 1
LRD
AW=    6, T6SK6LC:VW436
EU
S      AT6:Q0.5, 1
LRD
AW=    7, T6SK6LC:VW436
EU
S      AT7:Q0.6, 1
LRD
AW=    8, T6SK6LC:VW436
EU
S      AT8:Q0.7, 1
LPP
EU
S      #TAM6:L0.5, 1
Network 22
// SK6 TINH TG CHUONG
LD     #TAM6:L0.5
A      SM0.5
LD     T6RS:V11.7
CTU    T6SK6_TG:C42, 999
Network 23
// SK6 RESET CHUONG
// 
LDW>   T6SK6_TG:C42, T6SK6_TGD:VW438
EU
R      AT1:Q0.0, 8
R      T6SK6_TG:C42, 1
R      #TAM6:L0.5, 1
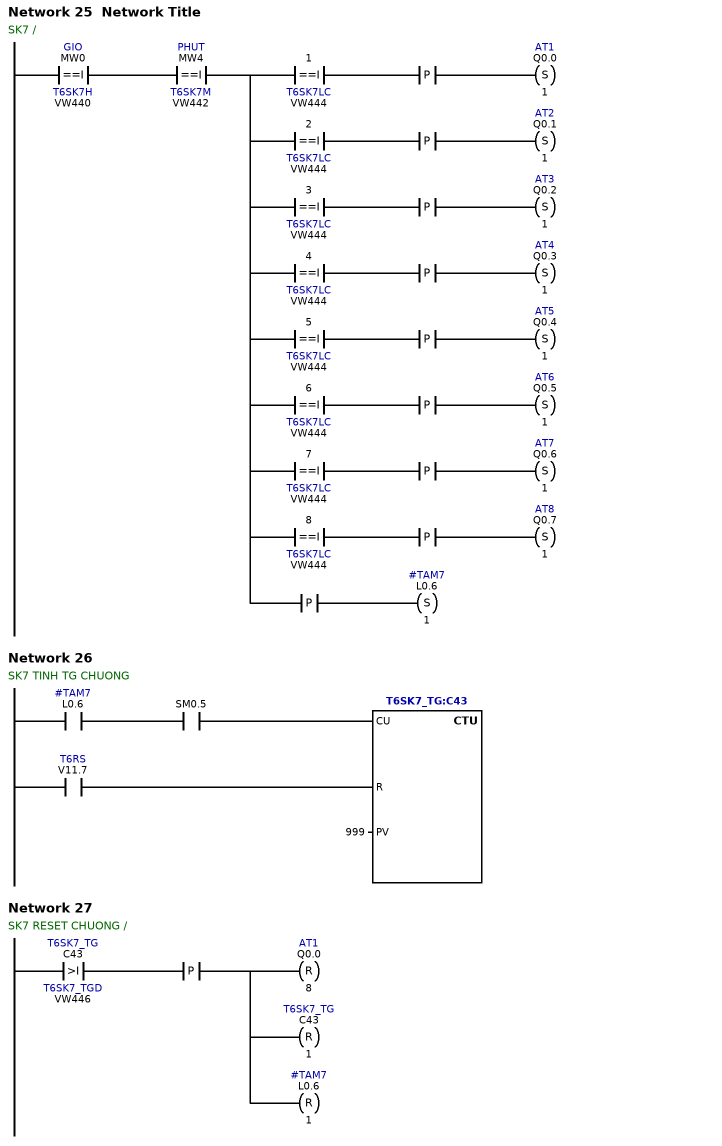
Network 25 // Network Title
// SK7
// 	
LDW=   GIO:MW0, T6SK7H:VW440
AW=    PHUT:MW4, T6SK7M:VW442
LPS
AW=    1, T6SK7LC:VW444
EU
S      AT1:Q0.0, 1
LRD
AW=    2, T6SK7LC:VW444
EU
S      AT2:Q0.1, 1
LRD
AW=    3, T6SK7LC:VW444
EU
S      AT3:Q0.2, 1
LRD
AW=    4, T6SK7LC:VW444
EU
S      AT4:Q0.3, 1
LRD
AW=    5, T6SK7LC:VW444
EU
S      AT5:Q0.4, 1
LRD
AW=    6, T6SK7LC:VW444
EU
S      AT6:Q0.5, 1
LRD
AW=    7, T6SK7LC:VW444
EU
S      AT7:Q0.6, 1
LRD
AW=    8, T6SK7LC:VW444
EU
S      AT8:Q0.7, 1
LPP
EU
S      #TAM7:L0.6, 1
Network 26
// SK7 TINH TG CHUONG
LD     #TAM7:L0.6
A      SM0.5
LD     T6RS:V11.7
CTU    T6SK7_TG:C43, 999
Network 27
// SK7 RESET CHUONG
// 
LDW>   T6SK7_TG:C43, T6SK7_TGD:VW446
EU
R      AT1:Q0.0, 8
R      T6SK7_TG:C43, 1
R      #TAM7:L0.6, 1
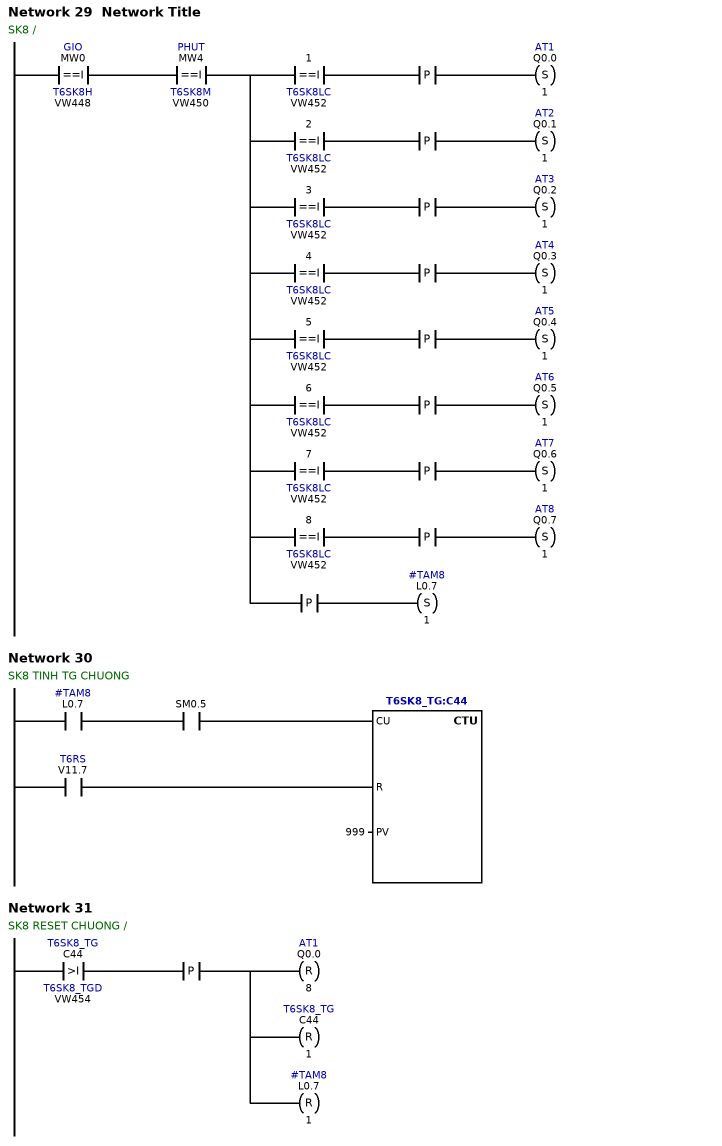
Network 29 // Network Title
// SK8
// 	
LDW=   GIO:MW0, T6SK8H:VW448
AW=    PHUT:MW4, T6SK8M:VW450
LPS
AW=    1, T6SK8LC:VW452
EU
S      AT1:Q0.0, 1
LRD
AW=    2, T6SK8LC:VW452
EU
S      AT2:Q0.1, 1
LRD
AW=    3, T6SK8LC:VW452
EU
S      AT3:Q0.2, 1
LRD
AW=    4, T6SK8LC:VW452
EU
S      AT4:Q0.3, 1
LRD
AW=    5, T6SK8LC:VW452
EU
S      AT5:Q0.4, 1
LRD
AW=    6, T6SK8LC:VW452
EU
S      AT6:Q0.5, 1
LRD
AW=    7, T6SK8LC:VW452
EU
S      AT7:Q0.6, 1
LRD
AW=    8, T6SK8LC:VW452
EU
S      AT8:Q0.7, 1
LPP
EU
S      #TAM8:L0.7, 1
Network 30
// SK8 TINH TG CHUONG
LD     #TAM8:L0.7
A      SM0.5
LD     T6RS:V11.7
CTU    T6SK8_TG:C44, 999
Network 31
// SK8 RESET CHUONG
// 
LDW>   T6SK8_TG:C44, T6SK8_TGD:VW454
EU
R      AT1:Q0.0, 8
R      T6SK8_TG:C44, 1
R      #TAM8:L0.7, 1
